// TIA Portal V17 export
// export: Created 2025-05-22T06:01:17.4374913Z, ExportSetting WithDefaults, DisplayName Totally Integrated Automation Portal, DisplayVersion V17 Update 8, DisplayName TIA Portal Openness, DisplayVersion V17 Update 8, DisplayName TIA Portal Version Control Interface, DisplayVersion V17, DisplayName SINAMICS Startdrive Advanced, DisplayVersion V17 SP2, DisplayName SINAMICS Startdrive G110M, G120, G120C, G120D, G120P, G115D, DisplayVersion V17 SP2, DisplayName SINAMICS Startdrive G130, G150, S120, S150, SINAMICS MV, S210, DisplayVersion V17 SP2, DisplayName STEP 7 Professional, DisplayVersion V17 Update 8, DisplayName SINUMERIK ONE STEP 7 Toolbox, DisplayVersion V17 Update 12, DisplayName SINUMERIK ONE PLC Basic Program Plus, DisplayVersion V17 Update 12, DisplayName SINUMERIK 840D sl STEP 7 Toolbox, DisplayVersion V17 Update 12, DisplayName STEP 7 Safety, DisplayVersion V17 Update 6, DisplayName WinCC Advanced, DisplayVersion V17 Update 8
DATA_BLOCK "DB16701_OPC_UA_MASTER_MACHINE_DATA_UPDATE_2"   // DB16702
{ S7_Optimized_Access := 'FALSE' }
VERSION : 0.1
// stored: AutoNumber false, DBAccessibleFromOPCUA true, DBAccessibleFromWebserver true, IsOnlyStoredInLoadMemory false, IsWriteProtectedInAS false
   VAR RETAIN
      GENERAL : Struct
         ID : Struct
            LINE : Int;   // Line ID
            MACHINE : Int;   // Machine ID
            PLC : Int;   // PLC ID
         END_STRUCT;
         "VERSION" : Struct
            MAJOR : Byte := 0;   // Major version
            MINOR : Byte := 2;   // Minor version
         END_STRUCT;
      END_STRUCT;
      PARAMS : Struct
         PART_TYPE : Int;   // Part type to be cladded
         UNIT_1 : Struct
            LASER : Struct
               BRIGHTLINE : Int;   // core ring intensity ratio
               BIFOCAL : Real;   // secondary/primary energy ratio
               POWER : Real;   // Laser power setpoint
               INJECTOR_DIAMETER : Real;   // inyectors diameter
               SPLITTER_TYPE : Array[1..40] of Char;   // splitter model reference
               NOZZLE_TYPE : Array[1..40] of Char;   // nozzle model reference
               NOZZLE_RADIAL_OFFSET : Real;   // nozzle radial adjust
               NOZZLE_TANGENTIAL_OFFSET : Real;   // nozzle tangential adjust
            END_STRUCT;
            MACHINE : Struct
               SHIELD_GAS_FLOW : Real;   // protection gas flow setpoint
               TANGENTIAL_SPEED : Real;   // tangential disc speed setpoint
               OVERLAP : Real;   // overlap setpoint
               LH_RADIAL_ANGLE : Real;   // laser radial angle
               LH_TANGENTIAL_ANGLE : Real;   // laser tangential angle
               LH_Z_POS : Real;   // heigh between part and nozzle
               CLADDING_SENSE : Bool;   // cladding sense 0 - from the inside out 1 - from the outside in
               STRATEGY : Bool;   // face order 0 - RN fist 1- NR first
               ST3_EXTRACTION_PRESSURE : Real;   // st3 extraction pressure setpoint
            END_STRUCT;
         END_STRUCT;
         UNIT_2 : Struct
            LASER : Struct
               BRIGHTLINE : Int;   // core ring intensity ratio
               BIFOCAL : Real;   // secondary/primary energy ratio
               POWER : Real;   // Laser power setpoint
               INJECTOR_DIAMETER : Real;   // inyectors diameter
               SPLITTER_TYPE : Array[1..40] of Char;   // splitter model reference
               NOZZLE_TYPE : Array[1..40] of Char;   // nozzle model reference
               NOZZLE_RADIAL_OFFSET : Real;   // nozzle radial adjust
               NOZZLE_TANGENTIAL_OFFSET : Real;   // nozzle tangential adjust
            END_STRUCT;
            MACHINE : Struct
               SHIELD_GAS_FLOW : Real;   // protection gas flow setpoint
               TANGENTIAL_SPEED : Real;   // tangential disc speed setpoint
               OVERLAP : Real;   // overlap setpoint
               LH_RADIAL_ANGLE : Real;   // laser head radial angle
               LH_TANGENTIAL_ANGLE : Real;   // laser head tangential angle
               LH_Z_POS : Real;   // heigh between part and nozzle
               CLADDING_SENSE : Bool;   // cladding sense 0 - from the inside out 1 - from the outside in
               STRATEGY : Bool;   // face order 0 - RN fist 1- NR first
               ST3_EXTRACTION_PRESSURE : Real;   // st3 extraction pressure setpoint
            END_STRUCT;
         END_STRUCT;
         EXTRACTION : Struct
            PRESSURE : Real;   // Extraction pressure setpoint
         END_STRUCT;
      END_STRUCT;
      MONITORING : Struct
         WORKER_ID : Int;
         EXTRACTION : Struct
            INPUT_KELLER_PRESSURE : Real;
            PRESSURE_DIFFERENCE_FILTER : Real;
         END_STRUCT;
         COOLING_SYSTEM : Struct
            INPUT_FLOW : Real;   // Entrada en máquina
            INPUT_TEMPERATURE : Real;   // Entrada en máquina
            OUTPUT_FLOW : Real;   // Salida de máquina
            OUTPUT_TEMPERATURE : Real;   // Salida de máquina
         END_STRUCT;
         UNIT_1 : Struct
            TEMPERATURE : Struct
               DISC_SURFACE : Real;   // disc surface temperature
               AMBIENT_PYROMETER : Real;   // pyrometer head internal temperature
            END_STRUCT;
            COOLING_SYSTEM : Struct
               LASER_HEAD_FLOW : Real;   // laser head cooling circuit flow
               LASER_HEAD_TEMPERATURE : Real;   // laser head cooling water output temperature
               LASER_FLOW : Real;   // laser source cooling circuit flow
               LASER_TEMPERATURE : Real;   // laser source cooling circuit temperature
               NOZZLE_FLOW : Real;   // powder nozzle cooling circuit flow
               NOZZLE_TEMPERATURE : Real;   // powder nozzle cooling circuit temperature
               SHIELD_FLOW : Real;   // shield cooling circuit flow
               SHIELD_TEMPERATURE : Real;   // shield cooling circuit temperature
            END_STRUCT;
            AIR_EXTRACTION : Struct
               OUTPUT_PRESSURE : Real;   // st3 extraction pressure
            END_STRUCT;
            CINEMATIC : Struct
               POSITIONS : Struct
                  CN : Struct
                     X13 : Real;   // X13 position
                     Z13 : Real;   // Z13 position
                  END_STRUCT;
               END_STRUCT;
               SPEED : Struct
                  X13 : Real;   // X13 speed
                  C13 : Real;   // C13 speed
               END_STRUCT;
            END_STRUCT;
            NOZZLE : Struct
               SHIELD_GAS_FLOW : Real;   // shielding gas flow
            END_STRUCT;
         END_STRUCT;
         UNIT_2 : Struct
            TEMPERATURE : Struct
               DISC_SURFACE : Real;   // disc surface temperature
               AMBIENT_PYROMETER : Real;   // pyrometer head internal temperature
            END_STRUCT;
            COOLING_SYSTEM : Struct
               LASER_HEAD_FLOW : Real;   // laser head cooling circuit flow
               LASER_HEAD_TEMPERATURE : Real;   // laser head cooling water output temperature
               LASER_FLOW : Real;   // laser source cooling circuit flow
               LASER_TEMPERATURE : Real;   // laser source cooling circuit temperature
               NOZZLE_FLOW : Real;   // powder nozzle cooling circuit flow
               NOZZLE_TEMPERATURE : Real;   // powder nozzle cooling circuit temperature
               SHIELD_FLOW : Real;   // shield cooling circuit flow
               SHIELD_TEMPERATURE : Real;   // shield cooling circuit temperature
            END_STRUCT;
            AIR_EXTRACTION : Struct
               OUTPUT_PRESSURE : Real;   // st3 extraction pressure
            END_STRUCT;
            CINEMATIC : Struct
               POSITIONS : Struct
                  CN : Struct
                     X23 : Real;   // X23 position
                     Z23 : Real;   // Z23 position
                  END_STRUCT;
               END_STRUCT;
               SPEED : Struct
                  X23 : Real;   // X23 speed
                  C23 : Real;   // C23 speed
               END_STRUCT;
            END_STRUCT;
            NOZZLE : Struct
               SHIELD_GAS_FLOW : Real;   // shielding gas flow
            END_STRUCT;
         END_STRUCT;
      END_STRUCT;
      STATUS : Struct
         ACK_BUTTON : Bool;
         PART_TRACKING : Struct
            DMC_U1_ST1 : Array[0..63] of Char;   // current DMC present in position
            DMC_U1_ST2 : Array[0..63] of Char;   // current DMC present in position
            DMC_U1_ST3 : Array[0..63] of Char;   // current DMC present in position
            DMC_U1_ST4 : Array[0..63] of Char;   // current DMC present in position
            DMC_U2_ST1 : Array[0..63] of Char;   // current DMC present in position
            DMC_U2_ST2 : Array[0..63] of Char;   // current DMC present in position
            DMC_U2_ST3 : Array[0..63] of Char;   // current DMC present in position
            DMC_U2_ST4 : Array[0..63] of Char;   // current DMC present in position
         END_STRUCT;
         MACHINE : Struct
            GLOBAL_STATUS : Int;   // 1-PRODUCING 2-WORKING 3-INACTIVE 4- MAINTENANCE 5-FAULTED
            CYCLE_ACTIVE : Int;   // 1- Continuous 2- single 3- robot dry 4- dry
            MODE_ACTIVE : Int;   // 1-auto 2- semiauto 3- manual
            HALF_LOAD : Bool;   // working with two fixtures (half load)
            SUBCYCLE : Struct
               RUN_OUT : Bool;   // Run out sequence active
               MANUAL_LOAD : Bool;   // loading part manually
               ROBOT_TEST : Bool;   // Robot test mode working
               CALIBRATION : Bool;   // Fixture calibration sequence active
               MASTER_MEAS : Bool;   // Measuring master part
            END_STRUCT;
            HW_DISABLE : Struct
               U1_PF : Bool;
               U2_PF : Bool;
               U1_ST3_MEAS : Bool;
               U1_ST3_COAX : Bool;
               U2_ST2_MEAS : Bool;
               U2_ST3_MEAS : Bool;
               U2_ST3_COAX : Bool;
               U3_NS : Bool;
               U3_RS : Bool;
               HOLA : Bool;
               U1_PYROMETER : Bool;
               U2_PYROMETER : Bool;
               U1_LASER : Bool;
               U2_LASER : Bool;
            END_STRUCT;
            PNEUMATIC : Struct
               ON : Bool;   // pneumatic on
               FAULTED : Bool;   // pneumatic faulted
            END_STRUCT;
         END_STRUCT;
         UNIT_1 : Struct
            FAULTED : Bool;   // Unit faulted
            ST0 : Struct
               FIXTURE_SEALED : Bool;   // Unit sealed
               TURNING : Bool;   // Fixtures turning
            END_STRUCT;
            ST1 : Struct
               FIXTURE_NUMBER : Int;   // fixture number present in station
               LOADING_PART : Bool;   // Robot loading part
               PART_PRESENT : Bool;   // Part present
               CLAMPING : Bool;   // Clamping part
               UNCLAMPING : Bool;   // Unclamping part
               MOTOR_RUNNING : Bool;   // motor running
            END_STRUCT;
            ST2 : Struct
               FIXTURE_NUMBER : Int;   // fixture number present in station
               MOTOR_RUNNING : Bool;   // motor running
            END_STRUCT;
            ST3 : Struct
               FIXTURE_NUMBER : Int;   // fixture number present in station
               SEALED : Bool;   // Station sealed
               CLADDING : Bool;   // cladding
               LIGHT_ON : Bool;   // light on
               MEASURING : Bool;   // perfilometer measuing part
               CALIBRATING : Bool;   // calibrating
               MOTOR_RUNNING : Bool;   // motor running
            END_STRUCT;
            ST4 : Struct
               FIXTURE_NUMBER : Int;   // fixture number present in station
               BLOW : Bool;   // Part blowing
               EXTRACTION_ON : Bool;   // extraction on
               SEALED : Bool;   // stations sealed
               MOTOR_RUNNING : Bool;   // motor running
            END_STRUCT;
            F1 : Struct
               CLAMPED : Bool;   // part clamped
               CALIBRATED_ST3 : Bool;   // calibration correct
            END_STRUCT;
            F2 : Struct
               CLAMPED : Bool;   // part clamped
               CALIBRATED_ST3 : Bool;   // calibration correct
            END_STRUCT;
            F3 : Struct
               CLAMPED : Bool;   // part clamped
               CALIBRATED_ST3 : Bool;   // calibration correct
            END_STRUCT;
            F4 : Struct
               CLAMPED : Bool;   // part clamped
               CALIBRATED_ST3 : Bool;   // calibration correct
            END_STRUCT;
            LASER : Struct
               PARKING : Bool;   // laser head at parking position
               PROGRAM_ACTIVE : Int;   // program active ID
            END_STRUCT;
         END_STRUCT;
         UNIT_2 : Struct
            FAULTED : Bool;   // Unit faulted
            ST0 : Struct
               FIXTURE_SEALED : Bool;   // Unit sealed
               TURNING : Bool;   // Fixtures turning
            END_STRUCT;
            ST1 : Struct
               FIXTURE_NUMBER : Int;   // fixture number present in station
               LOADING_PART : Bool;   // Robot loading part
               PART_PRESENT : Bool;   // Part present
               CLAMPING : Bool;   // Clamping part
               UNCLAMPING : Bool;   // Unclamping part
               MOTOR_RUNNING : Bool;   // motor running
            END_STRUCT;
            ST2 : Struct
               FIXTURE_NUMBER : Int;   // fixture number present in station
               MEASURING : Bool;   // perfilometer measuing part
               CALIBRATING : Bool;   // calibrating
               MOTOR_RUNNING : Bool;   // motor running
            END_STRUCT;
            ST3 : Struct
               FIXTURE_NUMBER : Int;   // fixture number present in station
               SEALED : Bool;   // Station sealed
               CLADDING : Bool;   // cladding
               LIGHT_ON : Bool;   // light on
               MEASURING : Bool;   // perfilometer measuing part
               CALIBRATING : Bool;   // calibrating
               MOTOR_RUNNING : Bool;   // motor running
            END_STRUCT;
            ST4 : Struct
               FIXTURE_NUMBER : Int;   // fixture number present in station
               BLOW : Bool;   // Part blowing
               EXTRACTION_ON : Bool;   // extraction on
               SEALED : Bool;   // stations sealed
               MOTOR_RUNNING : Bool;   // motor running
            END_STRUCT;
            F1 : Struct
               CLAMPED : Bool;   // part clamped
               CALIBRATED_ST2 : Bool;   // calibration correct
               CALIBRATED_ST3 : Bool;   // Calibrado realizado correctamente
            END_STRUCT;
            F2 : Struct
               CLAMPED : Bool;   // part clamped
               CALIBRATED_ST2 : Bool;   // calibration correct
               CALIBRATED_ST3 : Bool;   // calibration correct
            END_STRUCT;
            F3 : Struct
               CLAMPED : Bool;   // part clamped
               CALIBRATED_ST2 : Bool;   // calibration correct
               CALIBRATED_ST3 : Bool;   // calibration correct
            END_STRUCT;
            F4 : Struct
               CLAMPED : Bool;   // part clamped
               CALIBRATED_ST2 : Bool;   // calibration correct
               CALIBRATED_ST3 : Bool;   // calibration correct
            END_STRUCT;
            LASER : Struct
               PARKING : Bool;   // laser head at parking position
               PROGRAM_ACTIVE : Int;   // program active ID
            END_STRUCT;
         END_STRUCT;
         MEAS_STATION : Struct
            MEASURING : Bool;   // Measuring
            CALIBRATING : Bool;   // Calibratng measurement station
            MOTOR_RUNNING : Bool;   // motor running
            RS_CALIBRATED : Bool;   // Calibration correct
            NS_CALIBRATED : Bool;   // Calibration correct
         END_STRUCT;
         COOLING : Struct
            UNITS : Struct
               PUMP_ON : Bool;   // pump on
            END_STRUCT;
         END_STRUCT;
         EXTRACTION : Struct
            ON : Bool;   // Extraction running
            FAULTED : Bool;   // Extraction failed
         END_STRUCT;
      END_STRUCT;
      MAINTENANCE : Struct
         MAINT_EVENT : Struct
            REPLACEMENT : Bool;   // Replacement declared by worker
            UNIT_1 : Struct
               F1 : Bool;
               F2 : Bool;
               F3 : Bool;
               F4 : Bool;
               PROF_ST3 : Bool;
               PYROMETER : Bool;
               PYROMETER_EMISSIVITY : Real;
               CAM_ST3 : Bool;
               SEALING_ST3 : Bool;
               WATER_SYS : Bool;
               GAS_SYS : Bool;
               X : Bool;
               Z : Bool;
               C1 : Bool;
               C2 : Bool;
               C3 : Bool;
               C4 : Bool;
               "E" : Bool;
               LH : Bool;
               LH_RADIAL_ANGLE : Int;
               LH_TANGENTIAL_ANGLE : Int;
               LASER : Struct
                  PROCESS_GLASS : Bool;
                  FIBER_GLASS : Bool;
                  NOZZLE : Bool;
               END_STRUCT;
            END_STRUCT;
            UNIT_2 : Struct
               F1 : Bool;
               F2 : Bool;
               F3 : Bool;
               F4 : Bool;
               PROF_ST2 : Bool;
               PROF_ST3 : Bool;
               PYROMETER : Bool;
               PYROMETER_EMISSIVITY : Bool;
               CAM_ST3 : Bool;
               SEALING_ST3 : Bool;
               WATER_SYS : Bool;
               GAS_SYS : Bool;
               X : Bool;
               Z : Bool;
               C1 : Bool;
               C2 : Bool;
               C3 : Bool;
               C4 : Bool;
               "E" : Bool;
               LH : Bool;
               LH_RADIAL_ANGLE : Int;
               LH_TANGENTIAL_ANGLE : Int;
               LASER : Struct
                  PROCESS_GLASS : Bool;
                  FIBER_GLASS : Bool;
                  NOZZLE : Bool;
               END_STRUCT;
            END_STRUCT;
         END_STRUCT;
         MAINT_SEQ : Struct
            UNIT_1 : Struct
               PROFILOMETER_ST3 : Bool;
               CAMERA : Bool;
               REFERENCE : Bool;
               CONE_MEAS : Bool;
               LASER : Struct
                  PRIMES : Bool;
                  NOZZLE : Bool;
               END_STRUCT;
            END_STRUCT;
            UNIT_2 : Struct
               PROFILOMETER_ST2 : Bool;
               PROFILOMETER_ST3 : Bool;
               CAMERA : Bool;
               REFERENCE : Bool;
               CONE_MEAS : Bool;
               LASER : Struct
                  PRIMES : Bool;
                  NOZZLE : Bool;
               END_STRUCT;
            END_STRUCT;
         END_STRUCT;
      END_STRUCT;
      HOLA : Struct
         GENERAL : Struct
            ID : Struct
               LINE : Int;   // Line ID
               MACHINE : Int;   // Machine ID
               PLC : Int;   // PLC ID
            END_STRUCT;
            "VERSION" : Struct
               MAJOR : Byte := 0;   // Major version
               MINOR : Byte := 2;   // Minor version
            END_STRUCT;
         END_STRUCT;
         PARAMS : Struct
            PART_TYPE : Int;   // Part type to be cladded
            UNIT_1 : Struct
               LASER : Struct
                  BRIGHTLINE : Int;   // core ring intensity ratio
                  BIFOCAL : Real;   // secondary/primary energy ratio
                  POWER : Real;   // Laser power setpoint
                  INJECTOR_DIAMETER : Real;   // inyectors diameter
                  SPLITTER_TYPE : Array[1..40] of Char;   // splitter model reference
                  NOZZLE_TYPE : Array[1..40] of Char;   // nozzle model reference
                  NOZZLE_RADIAL_OFFSET : Real;   // nozzle radial adjust
                  NOZZLE_TANGENTIAL_OFFSET : Real;   // nozzle tangential adjust
               END_STRUCT;
               MACHINE : Struct
                  SHIELD_GAS_FLOW : Real;   // protection gas flow setpoint
                  TANGENTIAL_SPEED : Real;   // tangential disc speed setpoint
                  OVERLAP : Real;   // overlap setpoint
                  LH_RADIAL_ANGLE : Real;   // laser radial angle
                  LH_TANGENTIAL_ANGLE : Real;   // laser tangential angle
                  LH_Z_POS : Real;   // heigh between part and nozzle
                  CLADDING_SENSE : Bool;   // cladding sense 0 - from the inside out 1 - from the outside in
                  STRATEGY : Bool;   // face order 0 - RN fist 1- NR first
                  ST3_EXTRACTION_PRESSURE : Real;   // st3 extraction pressure setpoint
               END_STRUCT;
            END_STRUCT;
            UNIT_2 : Struct
               LASER : Struct
                  BRIGHTLINE : Int;   // core ring intensity ratio
                  BIFOCAL : Real;   // secondary/primary energy ratio
                  POWER : Real;   // Laser power setpoint
                  INJECTOR_DIAMETER : Real;   // inyectors diameter
                  SPLITTER_TYPE : Array[1..40] of Char;   // splitter model reference
                  NOZZLE_TYPE : Array[1..40] of Char;   // nozzle model reference
                  NOZZLE_RADIAL_OFFSET : Real;   // nozzle radial adjust
                  NOZZLE_TANGENTIAL_OFFSET : Real;   // nozzle tangential adjust
               END_STRUCT;
               MACHINE : Struct
                  SHIELD_GAS_FLOW : Real;   // protection gas flow setpoint
                  TANGENTIAL_SPEED : Real;   // tangential disc speed setpoint
                  OVERLAP : Real;   // overlap setpoint
                  LH_RADIAL_ANGLE : Real;   // laser head radial angle
                  LH_TANGENTIAL_ANGLE : Real;   // laser head tangential angle
                  LH_Z_POS : Real;   // heigh between part and nozzle
                  CLADDING_SENSE : Bool;   // cladding sense 0 - from the inside out 1 - from the outside in
                  STRATEGY : Bool;   // face order 0 - RN fist 1- NR first
                  ST3_EXTRACTION_PRESSURE : Real;   // st3 extraction pressure setpoint
               END_STRUCT;
            END_STRUCT;
            EXTRACTION : Struct
               PRESSURE : Real;   // Extraction pressure setpoint
            END_STRUCT;
         END_STRUCT;
         MONITORING : Struct
            WORKER_ID : Int;
            EXTRACTION : Struct
               INPUT_KELLER_PRESSURE : Real;
               PRESSURE_DIFFERENCE_FILTER : Real;
            END_STRUCT;
            COOLING_SYSTEM : Struct
               INPUT_FLOW : Real;   // Entrada en máquina
               INPUT_TEMPERATURE : Real;   // Entrada en máquina
               OUTPUT_FLOW : Real;   // Salida de máquina
               OUTPUT_TEMPERATURE : Real;   // Salida de máquina
            END_STRUCT;
            UNIT_1 : Struct
               TEMPERATURE : Struct
                  DISC_SURFACE : Real;   // disc surface temperature
                  AMBIENT_PYROMETER : Real;   // pyrometer head internal temperature
               END_STRUCT;
               COOLING_SYSTEM : Struct
                  LASER_HEAD_FLOW : Real;   // laser head cooling circuit flow
                  LASER_HEAD_TEMPERATURE : Real;   // laser head cooling water output temperature
                  LASER_FLOW : Real;   // laser source cooling circuit flow
                  LASER_TEMPERATURE : Real;   // laser source cooling circuit temperature
                  NOZZLE_FLOW : Real;   // powder nozzle cooling circuit flow
                  NOZZLE_TEMPERATURE : Real;   // powder nozzle cooling circuit temperature
                  SHIELD_FLOW : Real;   // shield cooling circuit flow
                  SHIELD_TEMPERATURE : Real;   // shield cooling circuit temperature
               END_STRUCT;
               AIR_EXTRACTION : Struct
                  OUTPUT_PRESSURE : Real;   // st3 extraction pressure
               END_STRUCT;
               CINEMATIC : Struct
                  POSITIONS : Struct
                     CN : Struct
                        X13 : Real;   // X13 position
                        Z13 : Real;   // Z13 position
                     END_STRUCT;
                  END_STRUCT;
                  SPEED : Struct
                     X13 : Real;   // X13 speed
                     C13 : Real;   // C13 speed
                  END_STRUCT;
               END_STRUCT;
               NOZZLE : Struct
                  SHIELD_GAS_FLOW : Real;   // shielding gas flow
               END_STRUCT;
            END_STRUCT;
            UNIT_2 : Struct
               TEMPERATURE : Struct
                  DISC_SURFACE : Real;   // disc surface temperature
                  AMBIENT_PYROMETER : Real;   // pyrometer head internal temperature
               END_STRUCT;
               COOLING_SYSTEM : Struct
                  LASER_HEAD_FLOW : Real;   // laser head cooling circuit flow
                  LASER_HEAD_TEMPERATURE : Real;   // laser head cooling water output temperature
                  LASER_FLOW : Real;   // laser source cooling circuit flow
                  LASER_TEMPERATURE : Real;   // laser source cooling circuit temperature
                  NOZZLE_FLOW : Real;   // powder nozzle cooling circuit flow
                  NOZZLE_TEMPERATURE : Real;   // powder nozzle cooling circuit temperature
                  SHIELD_FLOW : Real;   // shield cooling circuit flow
                  SHIELD_TEMPERATURE : Real;   // shield cooling circuit temperature
               END_STRUCT;
               AIR_EXTRACTION : Struct
                  OUTPUT_PRESSURE : Real;   // st3 extraction pressure
               END_STRUCT;
               CINEMATIC : Struct
                  POSITIONS : Struct
                     CN : Struct
                        X23 : Real;   // X23 position
                        Z23 : Real;   // Z23 position
                     END_STRUCT;
                  END_STRUCT;
                  SPEED : Struct
                     X23 : Real;   // X23 speed
                     C23 : Real;   // C23 speed
                  END_STRUCT;
               END_STRUCT;
               NOZZLE : Struct
                  SHIELD_GAS_FLOW : Real;   // shielding gas flow
               END_STRUCT;
            END_STRUCT;
         END_STRUCT;
         STATUS : Struct
            ACK_BUTTON : Bool;
            PART_TRACKING : Struct
               DMC_U1_ST1 : Array[0..63] of Char;   // current DMC present in position
               DMC_U1_ST2 : Array[0..63] of Char;   // current DMC present in position
               DMC_U1_ST3 : Array[0..63] of Char;   // current DMC present in position
               DMC_U1_ST4 : Array[0..63] of Char;   // current DMC present in position
               DMC_U2_ST1 : Array[0..63] of Char;   // current DMC present in position
               DMC_U2_ST2 : Array[0..63] of Char;   // current DMC present in position
               DMC_U2_ST3 : Array[0..63] of Char;   // current DMC present in position
               DMC_U2_ST4 : Array[0..63] of Char;   // current DMC present in position
            END_STRUCT;
            MACHINE : Struct
               GLOBAL_STATUS : Int;   // 1-PRODUCING 2-WORKING 3-INACTIVE 4- MAINTENANCE 5-FAULTED
               CYCLE_ACTIVE : Int;   // 1- Continuous 2- single 3- robot dry 4- dry
               MODE_ACTIVE : Int;   // 1-auto 2- semiauto 3- manual
               HALF_LOAD : Bool;   // working with two fixtures (half load)
               SUBCYCLE : Struct
                  RUN_OUT : Bool;   // Run out sequence active
                  MANUAL_LOAD : Bool;   // loading part manually
                  ROBOT_TEST : Bool;   // Robot test mode working
                  CALIBRATION : Bool;   // Fixture calibration sequence active
                  MASTER_MEAS : Bool;   // Measuring master part
               END_STRUCT;
               HW_DISABLE : Struct
                  U1_PF : Bool;
                  U2_PF : Bool;
                  U1_ST3_MEAS : Bool;
                  U1_ST3_COAX : Bool;
                  U2_ST2_MEAS : Bool;
                  U2_ST3_MEAS : Bool;
                  U2_ST3_COAX : Bool;
                  U3_NS : Bool;
                  U3_RS : Bool;
                  HOLA : Bool;
                  U1_PYROMETER : Bool;
                  U2_PYROMETER : Bool;
                  U1_LASER : Bool;
                  U2_LASER : Bool;
               END_STRUCT;
               PNEUMATIC : Struct
                  ON : Bool;   // pneumatic on
                  FAULTED : Bool;   // pneumatic faulted
               END_STRUCT;
            END_STRUCT;
            UNIT_1 : Struct
               FAULTED : Bool;   // Unit faulted
               ST0 : Struct
                  FIXTURE_SEALED : Bool;   // Unit sealed
                  TURNING : Bool;   // Fixtures turning
               END_STRUCT;
               ST1 : Struct
                  FIXTURE_NUMBER : Int;   // fixture number present in station
                  LOADING_PART : Bool;   // Robot loading part
                  PART_PRESENT : Bool;   // Part present
                  CLAMPING : Bool;   // Clamping part
                  UNCLAMPING : Bool;   // Unclamping part
                  MOTOR_RUNNING : Bool;   // motor running
               END_STRUCT;
               ST2 : Struct
                  FIXTURE_NUMBER : Int;   // fixture number present in station
                  MOTOR_RUNNING : Bool;   // motor running
               END_STRUCT;
               ST3 : Struct
                  FIXTURE_NUMBER : Int;   // fixture number present in station
                  SEALED : Bool;   // Station sealed
                  CLADDING : Bool;   // cladding
                  LIGHT_ON : Bool;   // light on
                  MEASURING : Bool;   // perfilometer measuing part
                  CALIBRATING : Bool;   // calibrating
                  MOTOR_RUNNING : Bool;   // motor running
               END_STRUCT;
               ST4 : Struct
                  FIXTURE_NUMBER : Int;   // fixture number present in station
                  BLOW : Bool;   // Part blowing
                  EXTRACTION_ON : Bool;   // extraction on
                  SEALED : Bool;   // stations sealed
                  MOTOR_RUNNING : Bool;   // motor running
               END_STRUCT;
               F1 : Struct
                  CLAMPED : Bool;   // part clamped
                  CALIBRATED_ST3 : Bool;   // calibration correct
               END_STRUCT;
               F2 : Struct
                  CLAMPED : Bool;   // part clamped
                  CALIBRATED_ST3 : Bool;   // calibration correct
               END_STRUCT;
               F3 : Struct
                  CLAMPED : Bool;   // part clamped
                  CALIBRATED_ST3 : Bool;   // calibration correct
               END_STRUCT;
               F4 : Struct
                  CLAMPED : Bool;   // part clamped
                  CALIBRATED_ST3 : Bool;   // calibration correct
               END_STRUCT;
               LASER : Struct
                  PARKING : Bool;   // laser head at parking position
                  PROGRAM_ACTIVE : Int;   // program active ID
               END_STRUCT;
            END_STRUCT;
            UNIT_2 : Struct
               FAULTED : Bool;   // Unit faulted
               ST0 : Struct
                  FIXTURE_SEALED : Bool;   // Unit sealed
                  TURNING : Bool;   // Fixtures turning
               END_STRUCT;
               ST1 : Struct
                  FIXTURE_NUMBER : Int;   // fixture number present in station
                  LOADING_PART : Bool;   // Robot loading part
                  PART_PRESENT : Bool;   // Part present
                  CLAMPING : Bool;   // Clamping part
                  UNCLAMPING : Bool;   // Unclamping part
                  MOTOR_RUNNING : Bool;   // motor running
               END_STRUCT;
               ST2 : Struct
                  FIXTURE_NUMBER : Int;   // fixture number present in station
                  MEASURING : Bool;   // perfilometer measuing part
                  CALIBRATING : Bool;   // calibrating
                  MOTOR_RUNNING : Bool;   // motor running
               END_STRUCT;
               ST3 : Struct
                  FIXTURE_NUMBER : Int;   // fixture number present in station
                  SEALED : Bool;   // Station sealed
                  CLADDING : Bool;   // cladding
                  LIGHT_ON : Bool;   // light on
                  MEASURING : Bool;   // perfilometer measuing part
                  CALIBRATING : Bool;   // calibrating
                  MOTOR_RUNNING : Bool;   // motor running
               END_STRUCT;
               ST4 : Struct
                  FIXTURE_NUMBER : Int;   // fixture number present in station
                  BLOW : Bool;   // Part blowing
                  EXTRACTION_ON : Bool;   // extraction on
                  SEALED : Bool;   // stations sealed
                  MOTOR_RUNNING : Bool;   // motor running
               END_STRUCT;
               F1 : Struct
                  CLAMPED : Bool;   // part clamped
                  CALIBRATED_ST2 : Bool;   // calibration correct
                  CALIBRATED_ST3 : Bool;   // Calibrado realizado correctamente
               END_STRUCT;
               F2 : Struct
                  CLAMPED : Bool;   // part clamped
                  CALIBRATED_ST2 : Bool;   // calibration correct
                  CALIBRATED_ST3 : Bool;   // calibration correct
               END_STRUCT;
               F3 : Struct
                  CLAMPED : Bool;   // part clamped
                  CALIBRATED_ST2 : Bool;   // calibration correct
                  CALIBRATED_ST3 : Bool;   // calibration correct
               END_STRUCT;
               F4 : Struct
                  CLAMPED : Bool;   // part clamped
                  CALIBRATED_ST2 : Bool;   // calibration correct
                  CALIBRATED_ST3 : Bool;   // calibration correct
               END_STRUCT;
               LASER : Struct
                  PARKING : Bool;   // laser head at parking position
                  PROGRAM_ACTIVE : Int;   // program active ID
               END_STRUCT;
            END_STRUCT;
            MEAS_STATION : Struct
               MEASURING : Bool;   // Measuring
               CALIBRATING : Bool;   // Calibratng measurement station
               MOTOR_RUNNING : Bool;   // motor running
               RS_CALIBRATED : Bool;   // Calibration correct
               NS_CALIBRATED : Bool;   // Calibration correct
            END_STRUCT;
            COOLING : Struct
               UNITS : Struct
                  PUMP_ON : Bool;   // pump on
               END_STRUCT;
            END_STRUCT;
            EXTRACTION : Struct
               ON : Bool;   // Extraction running
               FAULTED : Bool;   // Extraction failed
            END_STRUCT;
         END_STRUCT;
         MAINTENANCE : Struct
            MAINT_EVENT : Struct
               REPLACEMENT : Bool;   // Replacement declared by worker
               UNIT_1 : Struct
                  F1 : Bool;
                  F2 : Bool;
                  F3 : Bool;
                  F4 : Bool;
                  PROF_ST3 : Bool;
                  PYROMETER : Bool;
                  PYROMETER_EMISSIVITY : Real;
                  CAM_ST3 : Bool;
                  SEALING_ST3 : Bool;
                  WATER_SYS : Bool;
                  GAS_SYS : Bool;
                  X : Bool;
                  Z : Bool;
                  C1 : Bool;
                  C2 : Bool;
                  C3 : Bool;
                  C4 : Bool;
                  "E" : Bool;
                  LH : Bool;
                  LH_RADIAL_ANGLE : Int;
                  LH_TANGENTIAL_ANGLE : Int;
                  LASER : Struct
                     PROCESS_GLASS : Bool;
                     FIBER_GLASS : Bool;
                     NOZZLE : Bool;
                  END_STRUCT;
               END_STRUCT;
               UNIT_2 : Struct
                  F1 : Bool;
                  F2 : Bool;
                  F3 : Bool;
                  F4 : Bool;
                  PROF_ST2 : Bool;
                  PROF_ST3 : Bool;
                  PYROMETER : Bool;
                  PYROMETER_EMISSIVITY : Bool;
                  CAM_ST3 : Bool;
                  SEALING_ST3 : Bool;
                  WATER_SYS : Bool;
                  GAS_SYS : Bool;
                  X : Bool;
                  Z : Bool;
                  C1 : Bool;
                  C2 : Bool;
                  C3 : Bool;
                  C4 : Bool;
                  "E" : Bool;
                  LH : Bool;
                  LH_RADIAL_ANGLE : Int;
                  LH_TANGENTIAL_ANGLE : Int;
                  LASER : Struct
                     PROCESS_GLASS : Bool;
                     FIBER_GLASS : Bool;
                     NOZZLE : Bool;
                  END_STRUCT;
               END_STRUCT;
            END_STRUCT;
            MAINT_SEQ : Struct
               UNIT_1 : Struct
                  PROFILOMETER_ST3 : Bool;
                  CAMERA : Bool;
                  REFERENCE : Bool;
                  CONE_MEAS : Bool;
                  LASER : Struct
                     PRIMES : Bool;
                     NOZZLE : Bool;
                  END_STRUCT;
               END_STRUCT;
               UNIT_2 : Struct
                  PROFILOMETER_ST2 : Bool;
                  PROFILOMETER_ST3 : Bool;
                  CAMERA : Bool;
                  REFERENCE : Bool;
                  CONE_MEAS : Bool;
                  LASER : Struct
                     PRIMES : Bool;
                     NOZZLE : Bool;
                  END_STRUCT;
               END_STRUCT;
            END_STRUCT;
         END_STRUCT;
      END_STRUCT;
   END_VAR
BEGIN
END_DATA_BLOCK
